FUNCTION_BLOCK EL3121
VAR
	_io : EL3xx1_Data;
	{attribute addProperty Name "WcState"}
	_wcState : WcStateInputToggle;
	{attribute addProperty Name "Info data"}
	_infoData : InfoDataAds;
END_VAR

PROPERTY IO : REFERENCE TO EL3xx1_Data
GET
IO REF= _io;
END_GET
END_PROPERTY

PROPERTY WcState : REFERENCE TO WcStateInputToggle
GET
WcState REF= _wcState;
END_GET
END_PROPERTY

END_FUNCTION_BLOCK

(* stored: Version 1.1.0.1, ProductVersion 3.1.4024.9
   POU EL3121: Id {490a3cb9-18f1-0f72-204e-aceef53f37aa}, SpecialFunc None
   Property IO: Id {75be9566-7564-003e-168b-08e896434b73}
   Get Get: Id {58719f47-56a2-0583-1802-98020c97b17a}
   Property WcState: Id {248f52c8-a3e5-0301-0980-aa1bd365b8d5}
   Get Get: Id {2da04c00-abc6-0507-1b59-4b109c59817d} *)
